// ---- POUs/DALI/DALI_Setup/VISUs/Visu_DALICommissioning/Visu_Part102SetFading.TcVIS
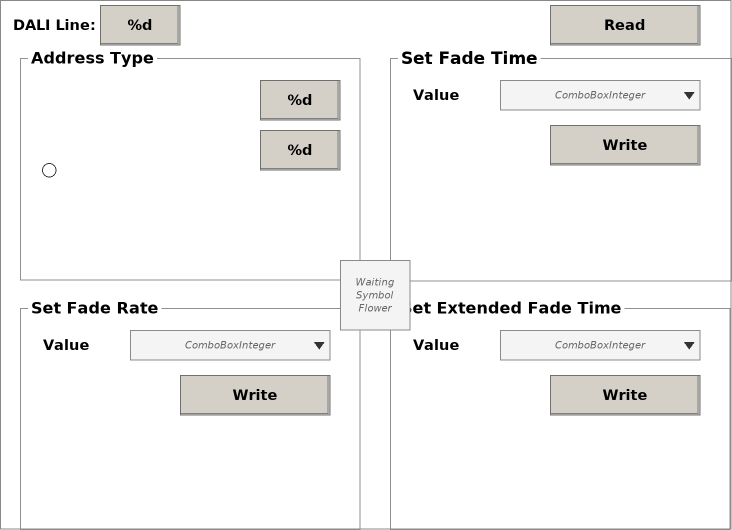
VISUALIZATION Visu_Part102SetFading  // 732x530
    GroupBox (390,50 342x231), "Set Fade Time"
        Textfield (20,30 100x30), "Value"
        ComboBoxInteger (110,30 200x30), variable: DALI_Commissioning.fbPart102SetFading.eFadeTime, text list: 'FadeTime'
        Button (160,75 150x40), "Write"
            OnMouseClick: execute { DALI_Commissioning.fbPart102SetFading.bWriteFadeTime := TRUE; }
    GroupBox (20,50 340x230), "Address Type"
        Button (240,30 80x40), "%d", text variable: DALI_Commissioning.fbPart102SetFading.nShortAddress
            OnMouseClick: write the text variable via Default, min 0, max 63, title "Insert Short Address"
        RadioButton (20,20 190x200), variable: DALI_Commissioning.fbPart102SetFading.eAddressType
            Areas[0]: Text=Short Address
            Areas[1]: Text=Group Address
            Areas[2]: Text=Broadcast
            Areas[3]: Text=Unaddressed
        Button (240,80 80x40), "%d", text variable: DALI_Commissioning.fbPart102SetFading.nGroupAddress
            OnMouseClick: write the text variable via Default, min 0, max 15, title "Insert Group Address"
    GroupBox (20,300 340x230), "Set Fade Rate"
        Textfield (20,30 100x30), "Value"
        ComboBoxInteger (110,30 200x30), variable: DALI_Commissioning.fbPart102SetFading.eFadeRate, text list: 'FadeRate'
        Button (160,75 150x40), "Write"
            OnMouseClick: execute { DALI_Commissioning.fbPart102setFading.bWriteFadeRate := TRUE; }
    GroupBox (390,300 340x230), "Set Extended Fade Time"
        Textfield (20,30 100x30), "Value"
        ComboBoxInteger (110,30 200x30), tooltip "Extended Fade Time only valid if Fade Time equals 0!", variable: DALI_Commissioning.fbPart102SetFading.eExtendedFadeTime, input disabled if: DALI_Commissioning.fbPart102SetFading.bNoFadeTime, text list: 'ExtendedFadeTime'
        Button (160,75 150x40), "Write", tooltip "Extended Fade Time only valid if Fade Time equals 0!", invisible if: DALI_Commissioning.fbPart102SetFading.bNoFadeTime, input disabled if: DALI_Commissioning.fbPart102SetFading.bNoFadeTime
            OnMouseClick: execute { DALI_Commissioning.fbPart102SetFading.bWriteExtendedFadeTime:=true; }
    Button (550,5 150x40), "Read", tooltip "Reads all Fading Parameters", invisible if: ( DALI_Commissioning.fbPart102SetFading.eAddressType >=1), input disabled if: ( DALI_Commissioning.fbPart102SetFading.eAddressType >=1)
        OnMouseClick: execute { DALI_Commissioning.fbPart102SetFading.bRead := TRUE; }
    WaitingSymbolFlower (340,260 70x70), invisible if: DALI_Commissioning.fbPart102SetFading.bHideWaitSymbol
    Group (10,5 170x40)
        Textfield (0,0 110x40), "DALI Line:"
        Button (90,0 80x40), "%d", text variable: GVL_Internal.nDALILine
            OnMouseClick: write the text variable via Default, min 1, max 10, title "Choose line"
END_VISUALIZATION

// ---- POUs/DALI/DALI_Setup/VISUs/Visu_DALICommissioning/Visu_Part103Addressing.TcVIS
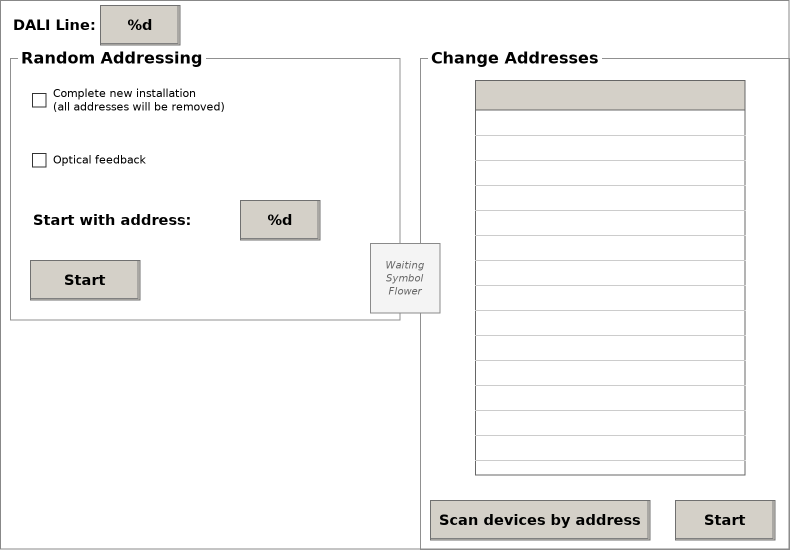
VISUALIZATION Visu_Part103Addressing  // 790x550
    GroupBox (420,50 370x500), "Change Addresses"
        Table (55,30 270x395), data array: DALI_Commissioning.fbPart103Addressing.aChangeAddressList
            p3854506369: DALI_Commissioning.fbPart103Addressing.aChangeAddressList[INDEX].nOldAddress
            p1892666644: DALI_Commissioning.fbPart103Addressing.aChangeAddressList[INDEX].nNewAddress
            p338671338: DALI_Commissioning.fbPart103Addressing.aChangeAddressList[INDEX].nRandomAddress
            p2170511999: DALI_Commissioning.fbPart103Addressing.aChangeAddressList[INDEX].nErrors
            Columns.Column.[0].Template: DALI_Commissioning.fbPart103Addressing.aNoShortAddress[INDEX]
            Columns.Column.[1].Template: DALI_Commissioning.fbPart103Addressing.aNoShortAddress[INDEX]; OnMouseClick: write the text variable via Default, min 0, max 63, title "New Short Address"
        Button (255,450 100x40), "Start"
            OnMouseClick: execute { DALI_Commissioning.fbPart103Addressing.bStartChangeAddress := TRUE; }
        Button (10,450 220x40), "Scan devices by address"
            OnMouseClick: execute { DALI_Commissioning.fbPart103Addressing.bScanDevices := TRUE; }
    GroupBox (10,50 390x270), "Random Addressing"
        Button (20,210 110x40), "Start"
            OnMouseClick: execute { DALI_Commissioning.fbPart103Addressing.bStartRandomAddressing := TRUE; }
        Checkbox (20,30 360x40), "Complete new installation (all addresses will be removed)", variable: DALI_Commissioning.fbPart103Addressing.bNewInstallation
        Checkbox (20,90 360x40), "Optical feedback", variable: DALI_Commissioning.fbPart103Addressing.bOpticalFeedback
        Textfield (20,150 200x40), "Start with address:"
        Button (230,150 80x40), "%d", text variable: DALI_Commissioning.fbPart103Addressing.nStartAddress
            OnMouseClick: write DALI_Commissioning.fbPart103Addressing.nStartAddress via Default, min 0, max 63, title "Insert Short Address"
    WaitingSymbolFlower (370,243 70x70), invisible if: DALI_Commissioning.fbPart103Addressing.bHideWaitSymbol
    Group (10,5 170x40)
        Textfield (0,0 110x40), "DALI Line:"
        Button (90,0 80x40), "%d", text variable: GVL_Internal.nDALILine
            OnMouseClick: write the text variable via Default, min 1, max 10, title "Choose line"
END_VISUALIZATION

// ---- POUs/DALI/DALI_Setup/VISUs/Visu_DALICommissioning/Visu_Part207.TcVIS
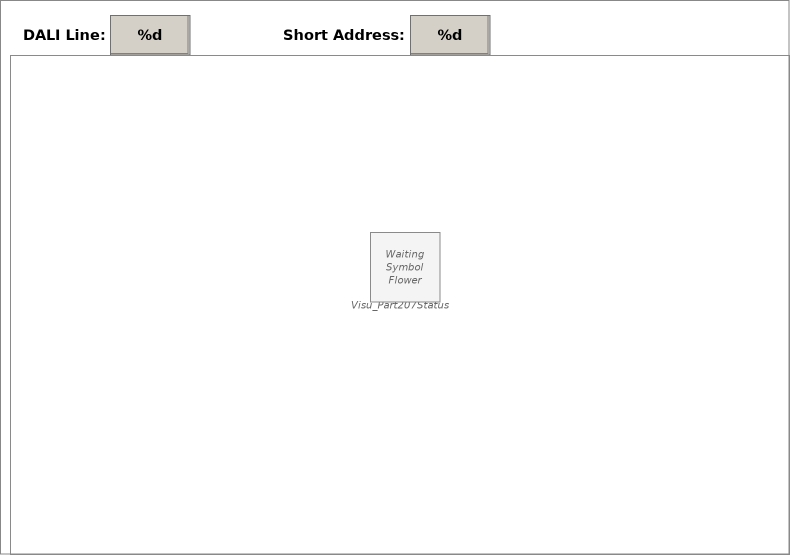
VISUALIZATION Visu_Part207  // 790x555
    Group (280,15 210x40)
        Textfield (0,0 130x40), "Short Address:"
        Button (130,0 80x40), "%d", text variable: DALI_Commissioning.fbPart207LED.nAddress
            OnMouseClick: write the text variable via Default, min 0, max 63, title "Insert Short Address"
    Group (20,15 170x40)
        Textfield (0,0 110x40), "DALI Line:"
        Button (90,0 80x40), "%d", text variable: GVL_Internal.nDALILine
            OnMouseClick: write the text variable via Default, min 1, max 10, title "Choose line"
    TabControl (10,55 780x500)
        shows Visu_Part207Status()
        shows Visu_Part207Parameters()
        shows Test()
        [0]: TabTitle=Status LED
        [1]: TabTitle=Parameters LED
        [2]: TabTitle=Paremeters LED
    WaitingSymbolFlower (370,232 70x70), invisible if: DALI_Commissioning.fbPart207LED.bHideWaitSymbol
END_VISUALIZATION

// ---- POUs/DALI/DALI_Setup/VISUs/Visu_DALICommissioning/Visu_Part207Status.TcVIS
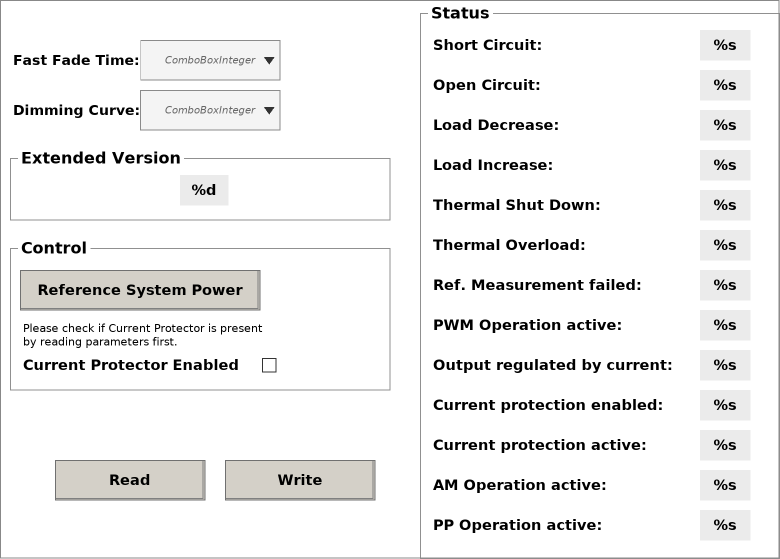
VISUALIZATION Visu_Part207Status  // 780x559
    GroupBox (420,5 360x554), "Status"
        Textfield (10,25 250x30), "Short Circuit:"
        Textfield (10,65 250x30), "Open Circuit:"
        Textfield (10,105 250x30), "Load Decrease:"
        Textfield (280,25 50x30), "%s", text variable: DALI_Commissioning.fbPart207LED.sShortCircuit
        Textfield (280,65 50x30), "%s", text variable: DALI_Commissioning.fbPart207LED.sOpenCircuit
        Textfield (280,105 50x30), "%s", text variable: DALI_Commissioning.fbPart207LED.sLoadDecrease
        Textfield (10,145 250x30), "Load Increase:"
        Textfield (280,145 50x30), "%s", text variable: DALI_Commissioning.fbPart207LED.sLoadIncrease
        Textfield (10,345 250x30), "Output regulated by current:", invisible if: DALI_Commissioning.fbPart207LED.bInvisible
        Textfield (10,385 250x30), "Current protection enabled:", invisible if: DALI_Commissioning.fbPart207LED.bInvisible
        Textfield (10,425 250x30), "Current protection active:", invisible if: DALI_Commissioning.fbPart207LED.bInvisible
        Textfield (10,185 250x30), "Thermal Shut Down:"
        Textfield (10,225 250x30), "Thermal Overload:"
        Textfield (10,265 250x30), "Ref. Measurement failed:"
        Textfield (10,465 250x30), "AM Operation active:", invisible if: DALI_Commissioning.fbPart207LED.bInvisible
        Textfield (10,505 250x30), "PP Operation active:", invisible if: DALI_Commissioning.fbPart207LED.bInvisible
        Textfield (10,305 250x30), "PWM Operation active:", invisible if: DALI_Commissioning.fbPart207LED.bInvisible
        Textfield (280,225 50x30), "%s", text variable: DALI_Commissioning.fbPart207LED.sThermalOverload
        Textfield (280,425 50x30), "%s", text variable: DALI_Commissioning.fbPart207LED.sCurrentProtectorActive, invisible if: DALI_Commissioning.fbPart207LED.bInvisible
        Textfield (280,385 50x30), "%s", text variable: DALI_Commissioning.fbPart207LED.sCurrentProtectorEnabled, invisible if: DALI_Commissioning.fbPart207LED.bInvisible
        Textfield (280,345 50x30), "%s", text variable: DALI_Commissioning.fbPart207LED.sOutputCurrentControlled, invisible if: DALI_Commissioning.fbPart207LED.bInvisible
        Textfield (280,465 50x30), "%s", text variable: DALI_Commissioning.fbPart207LED.sAMOperation, invisible if: DALI_Commissioning.fbPart207LED.bInvisible
        Textfield (280,505 50x30), "%s", text variable: DALI_Commissioning.fbPart207LED.sPowerPulseOperation, invisible if: DALI_Commissioning.fbPart207LED.bInvisible
        Textfield (280,265 50x30), "%s", text variable: DALI_Commissioning.fbPart207LED.sReferenceMeasurementFailed
        Textfield (280,185 50x30), "%s", text variable: DALI_Commissioning.fbPart207LED.sThermalShutDown
        Textfield (280,305 50x30), "%s", text variable: DALI_Commissioning.fbPart207LED.sPWMOperation, invisible if: DALI_Commissioning.fbPart207LED.bInvisible
    Button (225,460 150x40), "Write"
        OnMouseClick: execute { DALI_Commissioning.fbPart207LED.bWrite := TRUE; }
    GroupBox (10,240 380x150), "Control"
        Textfield (10,110 230x30), "Current Protector Enabled", invisible if: NOT DALI_Commissioning.fbPart207LED.bQueryCurrentProtectionDevicePresent
        Checkbox (250,110 30x30), variable: DALI_Commissioning.fbPart207LED.bCurrentProtector, invisible if: NOT DALI_Commissioning.fbPart207LED.bQueryCurrentProtectionDevicePresent, input disabled if: DALI_Commissioning.fbPart207LED.bQueryCurrentProtectionDevicePresent
        Button (10,30 240x40), "Reference System Power"
            OnMouseClick: execute { DALI_Commissioning.fbPart207LED.bReferenceSystempower := TRUE; }
        Label (10,80 300x30), "Please check if Current Protector is present by reading parameters first."
    Button (55,460 150x40), "Read"
        OnMouseClick: execute { DALI_Commissioning.fbPart207LED.bReadStatus := TRUE; }
    GroupBox (10,150 380x70), "Extended Version"
        Textfield (170,25 48x30), "%d", text variable: DALI_Commissioning.fbPart207LED.nExtendedVersionNumber
    Group (10,90 270x40)
        Textfield (0,0 130x40), "Dimming Curve:"
        ComboBoxInteger (130,0 140x40), variable: DALI_Commissioning.fbPart207LED.eDimmingCurve, text list: 'DimmingCurve'
    Group (10,40 270x40)
        ComboBoxInteger (130,0 140x40), variable: DALI_Commissioning.fbPart207LED.eFastFadeTime, text list: 'FastFadeTime'
        Textfield (0,0 130x40), "Fast Fade Time:"
END_VISUALIZATION

// ---- POUs/DALI/DALI_Setup/VISUs/Visu_DALICommissioning/Visu_Part300GenericDevice.TcVIS
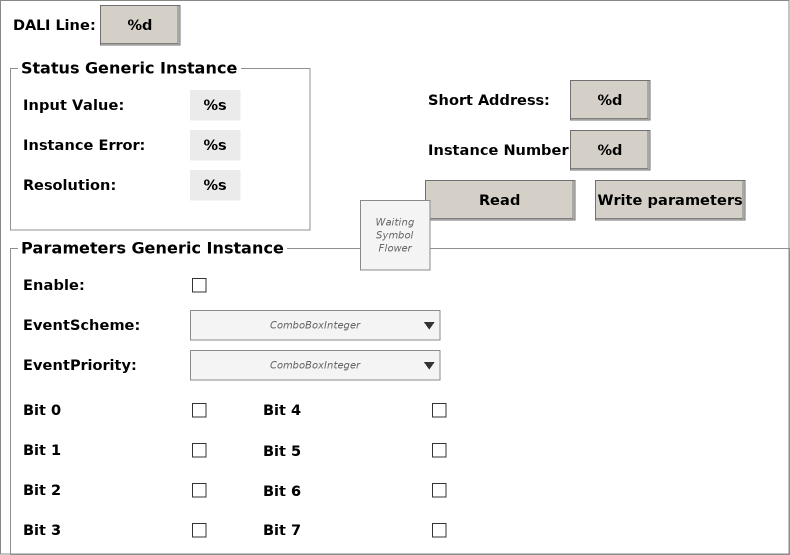
VISUALIZATION Visu_Part300GenericDevice  // 790x555
    GroupBox (10,240 780x315), "Parameters Generic Instance"
        Textfield (10,30 150x30), "Enable:"
        Checkbox (180,30 30x30), variable: DALI_Commissioning.fbPart300GenericDevice.bEnable
        Textfield (10,110 150x30), "EventPriority:"
        Textfield (10,195 100x30), "Bit 1"
        Textfield (10,155 100x30), "Bit 0"
        Checkbox (180,155 30x30), variable: DALI_Commissioning.fbPart300GenericDevice.bBit0
        Checkbox (180,195 30x30), variable: DALI_Commissioning.fbPart300GenericDevice.bBit1
        Textfield (10,235 100x30), "Bit 2"
        Textfield (250,155 100x30), "Bit 4"
        Textfield (250,196 100x30), "Bit 5"
        Checkbox (420,195 30x30), variable: DALI_Commissioning.fbPart300GenericDevice.bBit5
        Checkbox (420,155 30x30), variable: DALI_Commissioning.fbPart300GenericDevice.bBit4
        Checkbox (180,275 30x30), variable: DALI_Commissioning.fbPart300GenericDevice.bBit3
        Checkbox (180,235 30x30), variable: DALI_Commissioning.fbPart300GenericDevice.bBit2
        ComboBoxInteger (180,70 250x30), variable: DALI_Commissioning.fbPart300GenericDevice.eEventScheme, text list: 'EventScheme'
        Textfield (10,70 150x30), "EventScheme:"
        Textfield (250,236 100x30), "Bit 6"
        ComboBoxInteger (180,110 250x30), variable: DALI_Commissioning.fbPart300GenericDevice.eEventPriority, text list: 'EventPriority'
        Textfield (10,275 100x30), "Bit 3"
        Checkbox (420,235 30x30), variable: DALI_Commissioning.fbPart300GenericDevice.bBit6
        Checkbox (420,275 30x30), variable: DALI_Commissioning.fbPart300GenericDevice.bBit7
        Textfield (250,275 100x30), "Bit 7"
    GroupBox (10,60 300x170), "Status Generic Instance"
        Textfield (180,30 50x30), "%s", text variable: DALI_Commissioning.fbPart300GenericDevice.nInputValue
        Textfield (180,70 50x30), "%s", text variable: DALI_Commissioning.fbPart300GenericDevice.nInstanceError
        Textfield (180,110 50x30), "%s", text variable: DALI_Commissioning.fbPart300GenericDevice.nResolution
        Textfield (10,30 160x30), "Input Value:"
        Textfield (10,70 160x30), "Instance Error:"
        Textfield (10,110 160x30), "Resolution:"
    Button (425,180 150x40), "Read"
        OnMouseClick: execute { DALI_Commissioning.fbPart300GenericDevice.bRead := TRUE; }
    WaitingSymbolFlower (360,200 70x70), invisible if: DALI_Commissioning.fbPart300GenericDevice.bHideWaitSymbol
    Button (595,180 150x40), "Write parameters"
        OnMouseClick: execute { DALI_Commissioning.fbPart300GenericDevice.bWrite := TRUE; }
    Textfield (425,130 150x40), "Instance Number:"
    Textfield (425,80 150x40), "Short Address:"
    Button (570,80 80x40), "%d", text variable: DALI_Commissioning.fbPart300GenericDevice.nAddress
        OnMouseClick: write the text variable via Default, min 0, max 63, title "Insert Short Address"
    Button (570,130 80x40), "%d", text variable: DALI_Commissioning.fbPart300GenericDevice.nInstanceAddress
        OnMouseClick: write the text variable via Default, min 0, max 31, title "Insert instance number"
    Group (10,5 170x40)
        Textfield (0,0 110x40), "DALI Line:"
        Button (90,0 80x40), "%d", text variable: GVL_Internal.nDALILine
            OnMouseClick: write the text variable via Default, min 1, max 10, title "Choose line"
END_VISUALIZATION

// ---- POUs/DALI/DALI_Setup/VISUs/Visu_DALICommissioning/Visu_Part303OccupancySensor.TcVIS
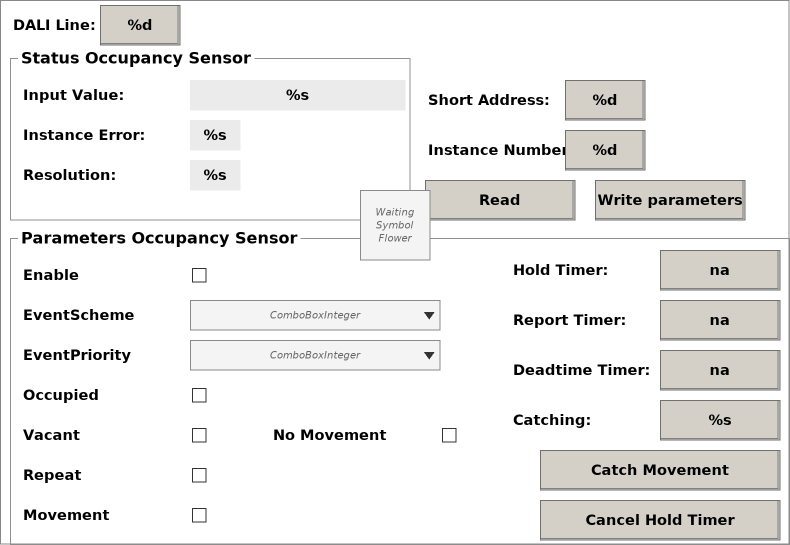
VISUALIZATION Visu_Part303OccupancySensor  // 790x545
    GroupBox (10,230 780x315), "Parameters Occupancy Sensor"
        Button (650,70 120x40), "%d s", text variable: DALI_Commissioning.fbPart303OccupancySensor.nReport
            OnMouseClick: write the text variable via Default, min 0, max 255, title "Insert value for report timer"
        Button (650,70 120x40), "na", invisible if: Not DALI_Commissioning.fbPart303OccupancySensor.bNoReportTimer, input disabled if: Not DALI_Commissioning.fbPart303OccupancySensor.bNoReportTimer
        Textfield (500,125 145x30), "Deadtime Timer:"
        Textfield (500,75 145x30), "Report Timer:"
        Textfield (500,25 145x30), "Hold Timer:"
        Button (650,20 120x40), "%d s", text variable: DALI_Commissioning.fbPart303OccupancySensor.nHold, invisible if: DALI_Commissioning.fbPart303OccupancySensor.bNoHoldTimer, input disabled if: DALI_Commissioning.fbPart303OccupancySensor.bNoHoldTimer
            OnMouseClick: write the text variable via Default, min 0, max 2538, title "Insert value for hold timer"
        Textfield (10,30 150x30), "Enable"
        Button (650,120 120x40), "%d ms", text variable: DALI_Commissioning.fbPart303OccupancySensor.nDeadtime
            OnMouseClick: write the text variable via Default, min 0, max 12750, title "Insert value for deadtime timer"
        Checkbox (180,30 30x30), variable: DALI_Commissioning.fbPart303OccupancySensor.bEnable
        Textfield (10,70 150x30), "EventScheme"
        Textfield (10,150 150x30), "Occupied"
        Textfield (10,190 150x30), "Vacant"
        Textfield (10,230 150x30), "Repeat"
        Textfield (10,270 150x30), "Movement"
        Textfield (260,190 150x30), "No Movement"
        Checkbox (180,150 30x30), variable: DALI_Commissioning.fbPart303OccupancySensor.bOccupied
        Checkbox (180,190 30x30), variable: DALI_Commissioning.fbPart303OccupancySensor.bVacant
        Checkbox (180,230 30x30), variable: DALI_Commissioning.fbPart303OccupancySensor.bRepeat
        Checkbox (430,190 30x30), variable: DALI_Commissioning.fbPart303OccupancySensor.bNoMovement
        ComboBoxInteger (180,70 250x30), variable: DALI_Commissioning.fbPart303OccupancySensor.eEventScheme, text list: 'EventScheme'
        Checkbox (180,270 30x30), variable: DALI_Commissioning.fbPart303OccupancySensor.bMovement
        Button (650,120 120x40), "na", invisible if: Not DALI_Commissioning.fbPart303OccupancySensor.bNoDeadtimeTimer, input disabled if: Not DALI_Commissioning.fbPart303OccupancySensor.bNoDeadtimeTimer
        Button (530,270 240x40), "Cancel Hold Timer"
            OnMouseClick: execute { DALI_Commissioning.fbPart303OccupancySensor.bCancelHoldTimer := true; }
        Textfield (10,110 150x30), "EventPriority"
        ComboBoxInteger (180,110 250x30), variable: DALI_Commissioning.fbPart303OccupancySensor.eEventPriority, text list: 'EventPriority'
        Button (650,20 120x40), "na", invisible if: Not DALI_Commissioning.fbPart303OccupancySensor.bNoHoldTimer, input disabled if: Not DALI_Commissioning.fbPart303OccupancySensor.bNoHoldTimer
        Button (530,220 240x40), "Catch Movement"
            OnMouseClick: execute { DALI_Commissioning.fbPart303OccupancySensor.bCatchMovement := true; }
        Textfield (500,175 145x30), "Catching:"
    GroupBox (10,50 400x170), "Status Occupancy Sensor"
        Textfield (10,30 160x30), "Input Value:"
        Textfield (10,70 160x30), "Instance Error:"
        Textfield (10,110 160x30), "Resolution:"
        Textfield (180,30 215x30), "%s", text variable: DALI_Commissioning.fbPart303OccupancySensor.sInputValue
        Textfield (180,70 50x30), "%s", text variable: DALI_Commissioning.fbPart303OccupancySensor.nInstanceError
        Textfield (180,110 50x30), "%s", text variable: DALI_Commissioning.fbPart303OccupancySensor.nResolution
    Button (425,180 150x40), "Read"
        OnMouseClick: execute { DALI_Commissioning.fbPart303OccupancySensor.bRead := TRUE; }
    WaitingSymbolFlower (360,190 70x70), invisible if: DALI_Commissioning.fbPart303OccupancySensor.bHideWaitSymbol
    Button (595,180 150x40), "Write parameters"
        OnMouseClick: execute { DALI_Commissioning.fbPart303OccupancySensor.bWrite := TRUE; }
    Button (660,400 120x40), "%s", text variable: DALI_Commissioning.fbPart303OccupancySensor.sCatching
        OnMouseClick: write the text variable via Default, min 0, max 12750, title "Insert value for deadtime timer"
    Group (10,5 170x40)
        Textfield (0,0 110x40), "DALI Line:"
        Button (90,0 80x40), "%d", text variable: GVL_Internal.nDALILine
            OnMouseClick: write the text variable via Default, min 1, max 10, title "Choose line"
    Textfield (425,80 130x40), "Short Address:"
    Button (565,80 80x40), "%d", text variable: DALI_Commissioning.fbPart303OccupancySensor.nAddress
        OnMouseClick: write the text variable via Default, min 0, max 63, title "Insert Short Address"
    Textfield (425,130 150x40), "Instance Number:"
    Button (565,130 80x40), "%d", text variable: DALI_Commissioning.fbPart303OccupancySensor.nInstanceAddress
        OnMouseClick: write the text variable via Default, min 0, max 31, title "Insert instance number"
END_VISUALIZATION
